// TIA Portal project "2022.06.08_移动指令的用法2" (V17)

(* hardware
DEVICE "S7-1200 station_1"  S7-1200 Station
   slot 0: "Rack_0"  S7-1200 Rack  Rack  V1.0
   slot 1: "PLC_1"  CPU 1212C DC/DC/DC  6ES7 212-1AE40-0XB0  V4.5
*)

// ===== PLC "PLC_1"  CPU 1212C DC/DC/DC =====

VAR_GLOBAL   // PLC tag table "默认变量表"
   "模拟量输入" AT %MW100 : Word;
   "Tag_3" AT %MW102 : UInt;
   "Tag_4" AT %MW104 : UInt;
   "Tag_5" AT %MW106 : UInt;
   "Tag_6" AT %I0.0 : Bool;
   "Tag_7" AT %M0.0 : Bool;
   "X(2)" AT %MW10 : Word;
   "Tag_9" AT %MW12 : UInt;
   "X" AT %MW0 : Word;
   "a" AT %MW2 : Word;
   "b" AT %MW4 : Int;
   "c" AT %MW8 : Int;
   "实时温度" AT %MD0 : Real;
   "Tag_10" AT %MD2 : Real;
   "f" AT %MD4 : Real;
   "g" AT %MD8 : Real;
   "X(1)" AT %MD12 : Real;
   "Tag_8" AT %MD16 : Real;
   "中间值(1)" AT %MD200 : Real;
   "中间值" AT %MD104 : Real;
   "工程值" AT %MD108 : Real;
   "要求的频率" AT %MD60 : Real;
   "百分比" AT %MD64 : Real;
   "Tag_12" AT %MW70 : Int;
   "Tag_2" AT %I0.1 : Bool;
   "0" AT %Q0.0 : Bool;
   "加热" AT %Q0.1 : Bool;
   "Tag_1" AT %MD100 : Time;
   "Tag_11" AT %M0.1 : Bool;
   "Tag_13" AT %QB0 : Byte;
   "Tag_14" AT %QB1 : Byte;
END_VAR

DATA_BLOCK "测试数据块_1"   // DB1
{ S7_Optimized_Access := 'FALSE' }
VERSION : 0.1
BEGIN
END_DATA_BLOCK

// folder: System blocks/Program resources

DATA_BLOCK "IEC_Timer_0_DB"   // DB2
{ S7_Optimized_Access := 'TRUE' }
AUTHOR : Simatic
FAMILY : IEC
NAME : IEC_TMR
VERSION : 1.0
// stored: InstanceOfName IEC_TIMER
"IEC_TIMER"
BEGIN
END_DATA_BLOCK

// folder: (top level)

ORGANIZATION_BLOCK "Main"   // OB1, LAD, ProgramCycle
TITLE = "Main Program Sweep (Cycle)"
{ S7_Optimized_Access := 'TRUE' }
VERSION : 0.1
   VAR_INPUT
      Initial_Call : Bool;   // Initial call of this OB
      Remanence : Bool;   // =True, if remanent data are available
   END_VAR
   VAR_TEMP   // added for the SCL form of the ladder/FBD networks
      _w1 : Bool;
   END_VAR
BEGIN

REGION Network 1
   // 切换成二进制，到头结束
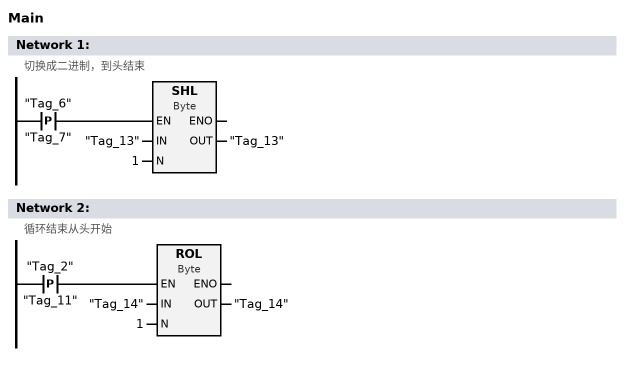
   RUNG wire#powerrail
      P_Contact(operand := "Tag_6", bit := "Tag_7")
      { S7_Templates := "SrcType := Byte" } Shl(in := "Tag_13", n := 1, out => "Tag_13")
   END_RUNG
   // the same network as SCL:
   #_w1 := "Tag_6" AND NOT "Tag_7";   // rising edge of "Tag_6"
   "Tag_7" := "Tag_6";
   IF #_w1 THEN "Tag_13" := SHL(IN := "Tag_13", N := 1); END_IF;
END_REGION

REGION Network 2
   // 循环结束从头开始
   #_w1 := "Tag_2" AND NOT "Tag_11";   // rising edge of "Tag_2"
   "Tag_11" := "Tag_2";
   IF #_w1 THEN "Tag_14" := ROL(IN := "Tag_14", N := 1); END_IF;
END_REGION
END_ORGANIZATION_BLOCK